RoboDK station: 2 - Pick and Place_solved.rdk

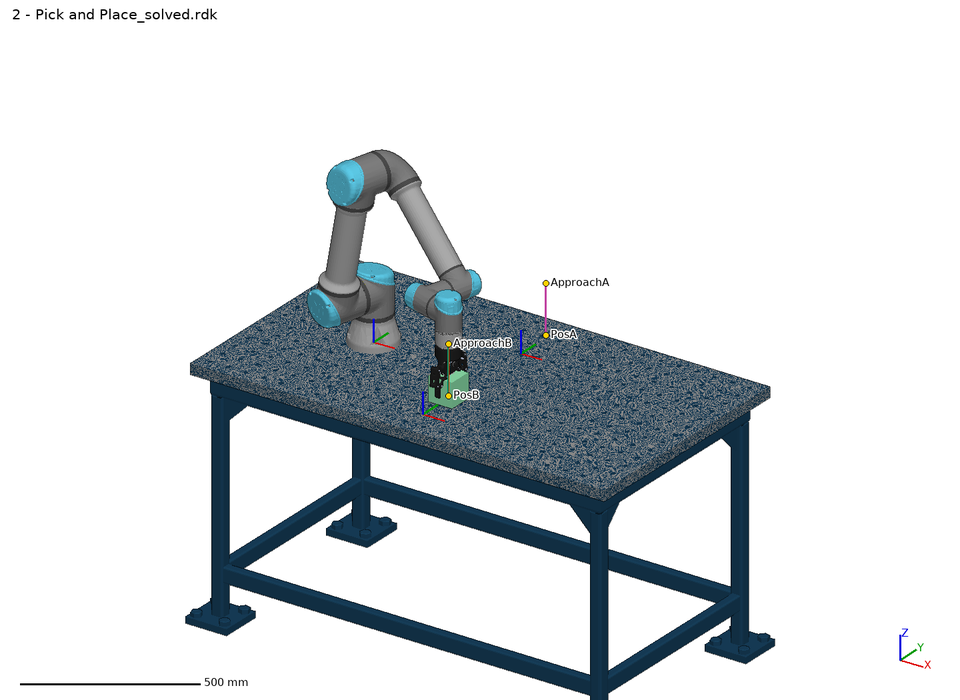
[picture v0: the station drawn from its stored meshes, robots at their saved joint values, targets as dots, program paths as lines]
Station 03A - Basic Pick and Place (saved by RoboDK 5.5.3). Poses are relative to the parent item; angles as X-Y-Z fixed-axis rotations.
Station parameters (name, value as stored): Palletizing Plugin
  - frame UR5e Base at (0, 0, 0) mm
    - robot UR5e: 6 axes, payload 5 kg, reach 850 mm, repeatability 0.03 mm, weight 18.4 kg
        modified DH rows (alpha deg, a mm, theta deg, d mm): 0, 0, 0, 162.5; 90, 0, 180, 0; 0, 425, 0, 0; 0, 392.25, 0, 133.3; -90, 0, 0, 99.7; 90, 0, 180, 99.6
        joint limits [-360, -360, -360, -360, -360, -360] to [360, 360, 360, 360, 360, 360]; home [0, -90, -90, -90, 90, 0]; saved at [-14.248, -101.954, -121.529, -46.517, 90, -14.248]
      - tool Gripper RobotiQ 85 Opened, TCP at (0, 0, 120) mm, size 147.4 x 146.8 x 75 mm
        - object box at (0, 0, 10) mm, rotated rx -180 ry 0 rz -90 deg, size 80 x 80 x 80 mm, geometry from box.sld
  - frame World at (0, 0, 0) mm
    - object Table at (0, 0, 0) mm, size 1420 x 820 x 800 mm, geometry from Table-1400x800x800.sld
  - frame PositionA at (375, 175, 0) mm
    - target ApproachA (Cartesian target) at (50, 50, 210) mm, rotated rx 180 ry 0 rz -90 deg; joints [43.99, -90.441, -113.295, -66.265, 90, 43.99] of UR5e
    - target PosA (Cartesian target) at (50, 50, 50) mm, rotated rx -180 ry 0 rz -90 deg; joints [43.99, -104.142, -124.633, -41.225, 90, 43.99] of UR5e
    - target Target 3 (Cartesian target) at (50, 50, 210) mm, rotated rx 180 ry 0 rz -90 deg; joints [43.99, -90.441, -113.295, -66.265, 90, 43.99] of UR5e
  - frame PositionB at (375, -295.45, 0) mm
    - target ApproachB (Cartesian target) at (50, 50, 210) mm, rotated rx 180 ry 0 rz -90 deg; joints [43.99, -90.441, -113.295, -66.265, 90, 43.99] of UR5e
    - target PosB (Cartesian target) at (50, 50, 50) mm, rotated rx -180 ry 0 rz -90 deg; joints [43.99, -104.142, -124.633, -41.225, 90, 43.99] of UR5e
  - program GripperOpen (1 instructions, listed below)
  - program GripperClose (1 instructions, listed below)
  - program PickA (6 instructions, listed below)
  - program PlaceB (6 instructions, listed below)
  - program PickB (5 instructions, listed below)
  - program PlaceA (6 instructions, listed below)
  - program MainProgram (4 instructions, listed below)
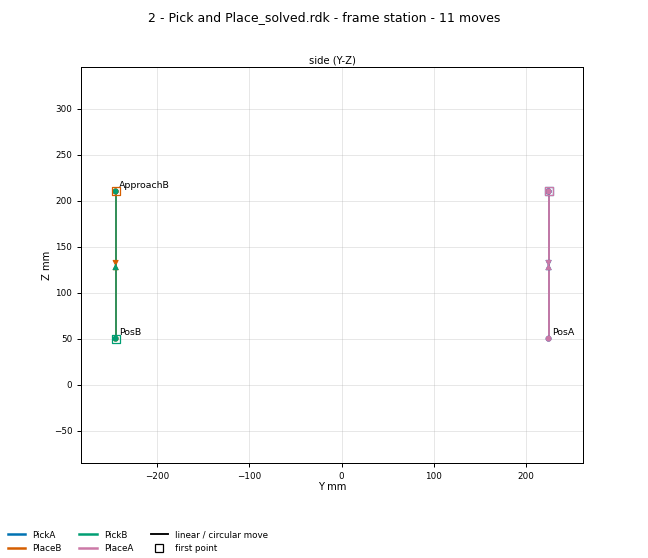
[picture p0: tool path of 2 - Pick and Place_solved.rdk in frame station, 11 of 11 moves have a stored position in this frame; points joined in program order, loops and branches not executed]

--- program GripperOpen (robot UR5e) ---
  Detach from Gripper RobotiQ 85 Opened

--- program GripperClose (robot UR5e) ---
  Attach to Gripper RobotiQ 85 Opened

--- program PickA (robot UR5e) ---
  Set Ref.: PositionA
  Set Tool: Gripper RobotiQ 85 Opened
  MoveJ (ApproachA)
  MoveL (PosA)
  Call GripperClose
  MoveL (ApproachA)

--- program PlaceB (robot UR5e) ---
  Set Ref.: PositionB
  Set Tool: Gripper RobotiQ 85 Opened
  MoveJ (ApproachB)
  MoveL (PosB)
  Call GripperOpen
  MoveL (ApproachB)

--- program PickB (robot UR5e) ---
  Set Ref.: PositionB
  Set Tool: Gripper RobotiQ 85 Opened
  MoveL (PosB)
  Call GripperClose
  MoveL (ApproachB)

--- program PlaceA (robot UR5e) ---
  Set Ref.: PositionA
  Set Tool: Gripper RobotiQ 85 Opened
  MoveJ (ApproachA)
  MoveL (PosA)
  Call GripperOpen
  MoveL (ApproachA)

--- program MainProgram (robot UR5e) ---
  Call PickA
  Call PlaceB
  Call PickB
  Call PlaceA
